TYPE ST_BaseControlElement_Homing :
STRUCT
	cmdExecute				: FB_BaseCommand;
	bIsNeeded				: BOOL := TRUE;		//pamieta czy juz element został wybazowany na początku true po bazowaniu zostaje ustawione na false
	bWithoutHoming			: BOOL;				//ustawienie czy ma być bazowanie czy nie
	iElementHomingStep		: INT;
END_STRUCT
END_TYPE

(* stored: Version 1.1.0.1
   DUT ST_BaseControlElement_Homing: Id {e14af5fb-2b04-0472-3dbe-debdd0bcf998} *)
